FUNCTION_BLOCK TowParametersSelector (* Basic Function Block Type *)
  (* Standard: 61499-2 *)
  (* Version 0.0, 7/3/2024, SESA713705, Schneider Electric, Template *)
  PACKAGE SE.Nereda;
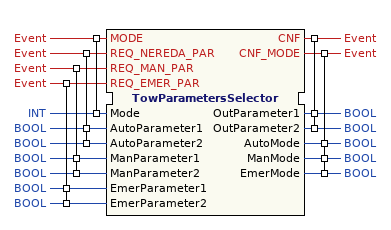
  EVENT_INPUT
    MODE WITH Mode;
    REQ_NEREDA_PAR WITH AutoParameter1, AutoParameter2;
    REQ_MAN_PAR WITH ManParameter1, ManParameter2;
    REQ_EMER_PAR WITH EmerParameter2, EmerParameter1;
  END_EVENT
  EVENT_OUTPUT
    CNF WITH OutParameter1, OutParameter2; (* Execution Confirmation *)
    CNF_MODE WITH ManMode, AutoMode, EmerMode;
  END_EVENT
  VAR_INPUT
    Mode : INT;
    AutoParameter1 : BOOL;
    AutoParameter2 : BOOL;
    ManParameter1 : BOOL;
    ManParameter2 : BOOL;
    EmerParameter1 : BOOL;
    EmerParameter2 : BOOL;
  END_VAR
  VAR_OUTPUT
    OutParameter1 : BOOL;
    OutParameter2 : BOOL;
    AutoMode : BOOL;
    ManMode : BOOL;
    EmerMode : BOOL;
  END_VAR
  VAR
    InParameter1 : BOOL;
    InParameter2 : BOOL;
  END_VAR
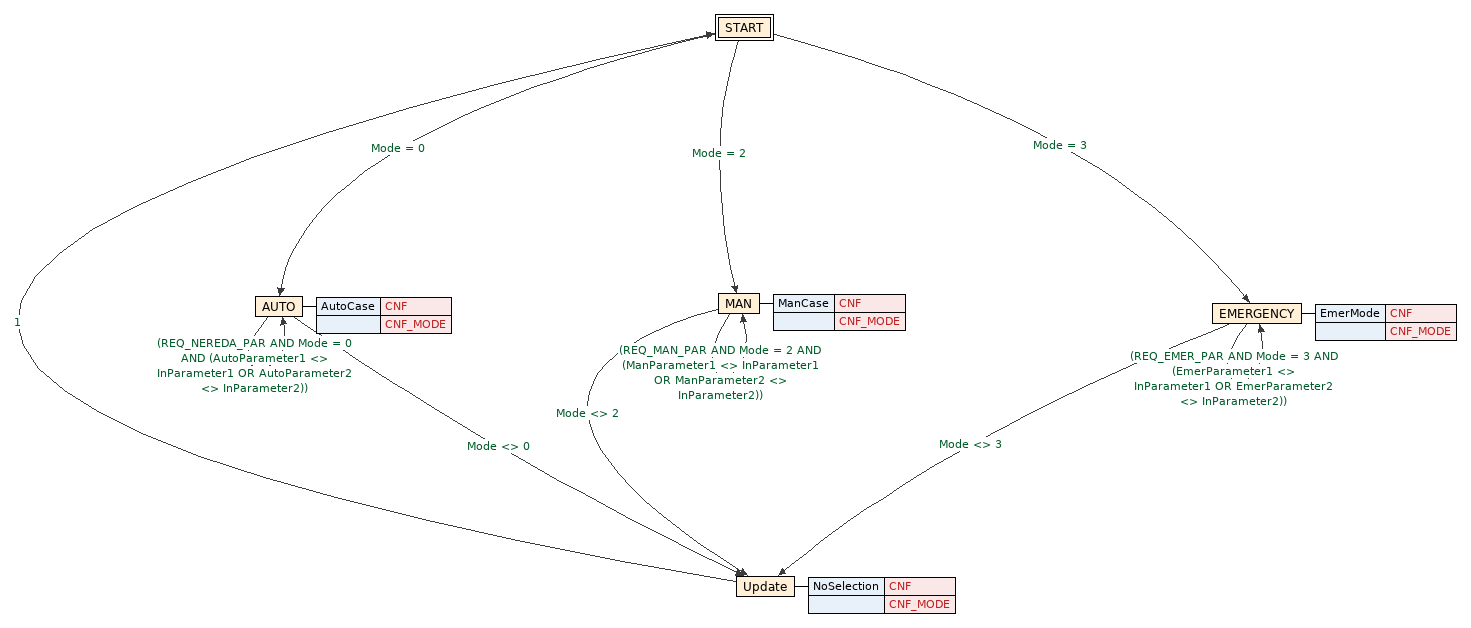
  EC_STATES
    START; (* Initial State *)
    AUTO : AutoCase -> CNF, -> CNF_MODE;
    MAN : ManCase -> CNF, -> CNF_MODE;
    EMERGENCY : EmerMode -> CNF, -> CNF_MODE;
    Update : NoSelection -> CNF, -> CNF_MODE;
  END_STATES
  EC_TRANSITIONS
    START TO AUTO := Mode = 0;
    START TO MAN := Mode = 2;
    AUTO TO AUTO := (REQ_NEREDA_PAR AND Mode = 0 AND (AutoParameter1 <> InParameter1 OR AutoParameter2 <> InParameter2));
    MAN TO MAN := (REQ_MAN_PAR AND Mode = 2 AND (ManParameter1 <> InParameter1 OR ManParameter2 <> InParameter2));
    START TO EMERGENCY := Mode = 3;
    EMERGENCY TO EMERGENCY := (REQ_EMER_PAR AND Mode = 3 AND (EmerParameter1 <> InParameter1 OR EmerParameter2 <> InParameter2));
    Update TO START := 1;
    MAN TO Update := Mode <> 2;
    AUTO TO Update := Mode <> 0;
    EMERGENCY TO Update := Mode <> 3;
  END_TRANSITIONS
  ALGORITHM AutoCase IN ST:
;

OutParameter1 := AutoParameter1;
OutParameter2 := AutoParameter2;
InParameter1 := AutoParameter1;
InParameter2 := AutoParameter2;

AutoMode := TRUE;
ManMode := FALSE;
EmerMode := FALSE;
  END_ALGORITHM
  ALGORITHM ManCase IN ST:
;

OutParameter1 := ManParameter1;
OutParameter2 := ManParameter2;
InParameter1 := ManParameter1;
InParameter2 := ManParameter2;

AutoMode := FALSE;
ManMode := TRUE;
EmerMode := FALSE;
  END_ALGORITHM
  ALGORITHM EmerMode IN ST:
;
OutParameter1 := EmerParameter1;
OutParameter2 := EmerParameter2;
InParameter1 := EmerParameter1;
InParameter2 := EmerParameter2;

AutoMode := FALSE;
ManMode := FALSE;
EmerMode := TRUE;
  END_ALGORITHM
  ALGORITHM NoSelection IN ST:
;
OutParameter1 := FALSE;
OutParameter2 := FALSE;
InParameter1 := FALSE;
InParameter2 := FALSE;
AutoMode := FALSE;
ManMode := FALSE;
EmerMode := FALSE;
  END_ALGORITHM
END_FUNCTION_BLOCK
